Omron CX-Programmer project NewProject (CX-Programmer 9.73)

# PLC NewPLC1: CP1L M

## Global symbols (name address type ; comment)
100.12 BOOL  ; INDIKATOR_AKHIR
0.02 BOOL  ; S_ADONAN
100.01 BOOL  ; GULA
0.00 BOOL  ; PB START
0.01 BOOL  ; S_KUNTELUR
0.03 BOOL  ; S_CETAK
0.04 BOOL  ; S_TOPPING
0.05 BOOL  ; S_AKHIR
100.00 BOOL  ; TEPUNG
100.02 BOOL  ; RAGI
100.03 BOOL  ; SUSU
100.04 BOOL  ; KUNING_TELUR
100.05 BOOL  ; MINYAK
100.06 BOOL  ; GARAM
100.07 BOOL  ; AIR
100.08 BOOL  ; MIXER
100.09 BOOL  ; INDIKATOR_ADONAN
100.10 BOOL  ; CONVEYOR
100.11 BOOL  ; TOPPING
C0000 BOOL  ; KUNING TELUR
C0001 BOOL  ; CETAKAN_DONAT
T0000 BOOL  ; TEPUNG
T0001 BOOL  ; GULA PASIR
T0002 BOOL  ; RAGI
T0003 BOOL  ; SUSU
T0004 BOOL  ; MINYAK
T0005 BOOL  ; GARAM
T0006 BOOL  ; AIR
T0007 BOOL  ; MIXER
T0011 BOOL  ; TOPPING

## Program NewProgram1 (cyclic task 0)
Local symbols
CT5 BOOL

### Section Section1

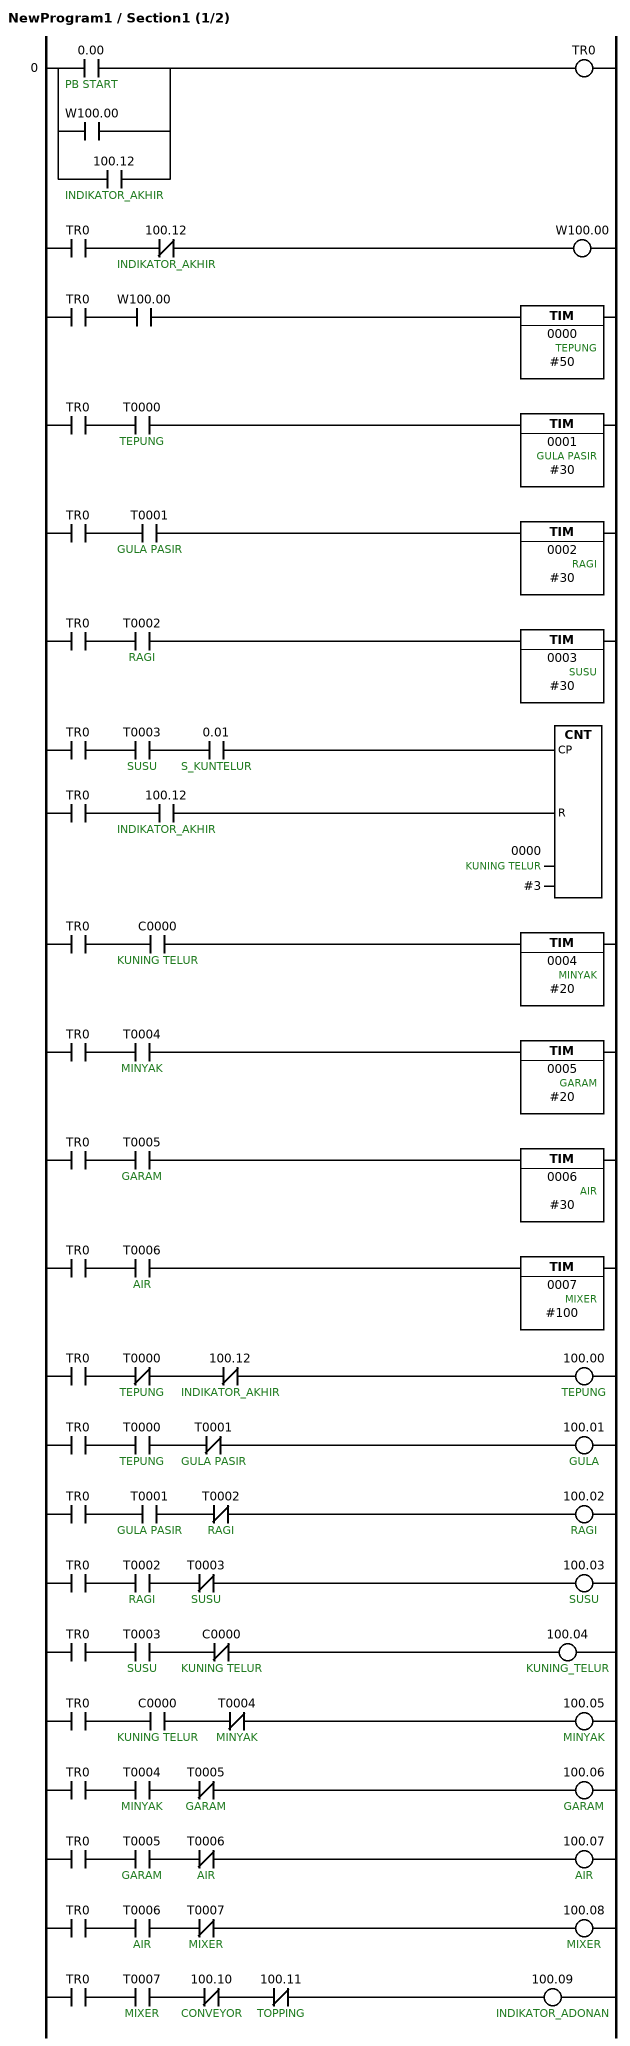
; rung 0
LD 0.00  ; PB START
OR W100.00
OR 100.12  ; INDIKATOR_AKHIR
OUT TR0
ANDNOT 100.12  ; INDIKATOR_AKHIR
OUT W100.00
LD TR0
AND W100.00
TIM 0000 #50  ; TEPUNG
LD TR0
AND T0000  ; TEPUNG
TIM 0001 #30  ; GULA PASIR
LD TR0
AND T0001  ; GULA PASIR
TIM 0002 #30  ; RAGI
LD TR0
AND T0002  ; RAGI
TIM 0003 #30  ; SUSU
LD TR0
AND T0003  ; SUSU
AND 0.01  ; S_KUNTELUR
LD TR0
AND 100.12  ; INDIKATOR_AKHIR
CNT 0000 #3  ; KUNING TELUR
LD TR0
AND C0000  ; KUNING TELUR
TIM 0004 #20  ; MINYAK
LD TR0
AND T0004  ; MINYAK
TIM 0005 #20  ; GARAM
LD TR0
AND T0005  ; GARAM
TIM 0006 #30  ; AIR
LD TR0
AND T0006  ; AIR
TIM 0007 #100  ; MIXER
LD TR0
ANDNOT T0000  ; TEPUNG
ANDNOT 100.12  ; INDIKATOR_AKHIR
OUT 100.00  ; TEPUNG
LD TR0
AND T0000  ; TEPUNG
ANDNOT T0001  ; GULA PASIR
OUT 100.01  ; GULA
LD TR0
AND T0001  ; GULA PASIR
ANDNOT T0002  ; RAGI
OUT 100.02  ; RAGI
LD TR0
AND T0002  ; RAGI
ANDNOT T0003  ; SUSU
OUT 100.03  ; SUSU
LD TR0
AND T0003  ; SUSU
ANDNOT C0000  ; KUNING TELUR
OUT 100.04  ; KUNING_TELUR
LD TR0
AND C0000  ; KUNING TELUR
ANDNOT T0004  ; MINYAK
OUT 100.05  ; MINYAK
LD TR0
AND T0004  ; MINYAK
ANDNOT T0005  ; GARAM
OUT 100.06  ; GARAM
LD TR0
AND T0005  ; GARAM
ANDNOT T0006  ; AIR
OUT 100.07  ; AIR
LD TR0
AND T0006  ; AIR
ANDNOT T0007  ; MIXER
OUT 100.08  ; MIXER
LD TR0
AND T0007  ; MIXER
ANDNOT 100.10  ; CONVEYOR
ANDNOT 100.11  ; TOPPING
OUT 100.09  ; INDIKATOR_ADONAN

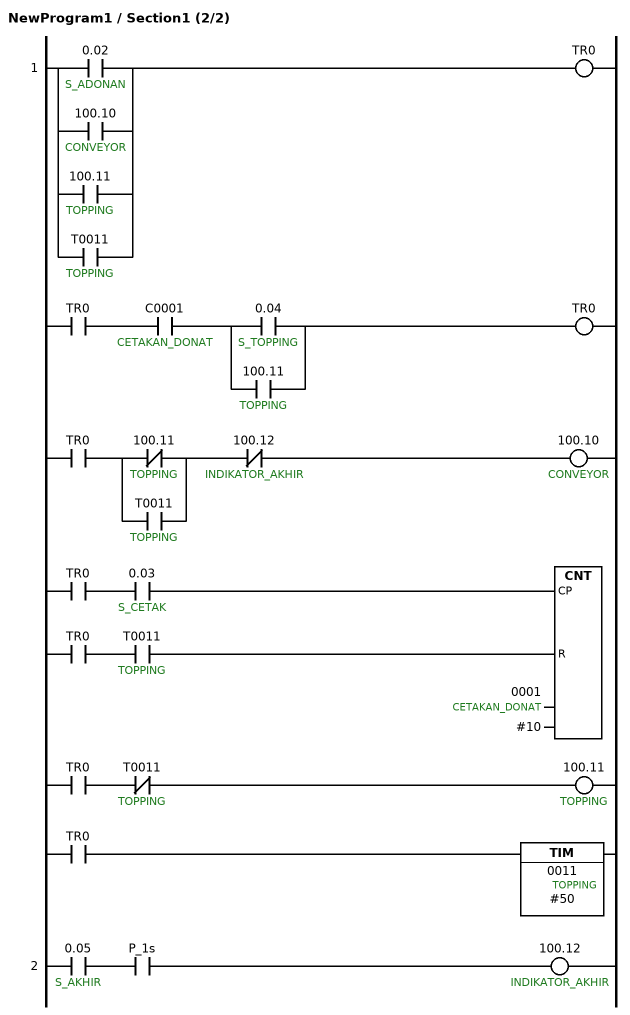
; rung 1
LD 0.02  ; S_ADONAN
OR 100.10  ; CONVEYOR
OR 100.11  ; TOPPING
OR T0011  ; TOPPING
OUT TR0
LDNOT 100.11  ; TOPPING
OR T0011  ; TOPPING
ANDLD
ANDNOT 100.12  ; INDIKATOR_AKHIR
OUT 100.10  ; CONVEYOR
LD TR0
AND 0.03  ; S_CETAK
LD TR0
AND T0011  ; TOPPING
CNT 0001 #10  ; CETAKAN_DONAT
LD TR0
AND C0001  ; CETAKAN_DONAT
LD 0.04  ; S_TOPPING
OR 100.11  ; TOPPING
ANDLD
OUT TR0
ANDNOT T0011  ; TOPPING
OUT 100.11  ; TOPPING
LD TR0
TIM 0011 #50  ; TOPPING
; rung 2
LD 0.05  ; S_AKHIR
AND P_1s
OUT 100.12  ; INDIKATOR_AKHIR

### Section END
; rung 0
END(001)